Fanuc KAREL source: kt00002.KL

PROGRAM KT00002
%NOLOCKGROUP
VAR
I1:INTEGER;I2:INTEGER;OUT:REAL
BEGIN
--
--
I1=2
I2=3
I1=2
I2=3
OUT=((I1+I2))
END KT00002
